PROGRAM CycleTest
VAR
	bCycleStart1:BOOL:= FALSE;
	bCycleStart2:BOOL:= FALSE;
	LevelToStart:INT:=3;
	iLevel:INT:=1;
	iNoOfLevel:INT:=4; //NO_OF_LEVEL;
	nState:INT;
	nCount:INT:=1;
	fbGUI_TEST : ARRAY [1..NO_OF_LEVEL] OF FB_GUI_TEST;
	arrLevelStartBits :ARRAY[1..NO_OF_LEVEL] OF BOOL;
	
	TDelay : TON;
	TDelay1: TON;
	TDelay2 : TON;
	ClearTCSEvent: TON;
	tCaptureDelay: TIME:= T#1000MS;
	tDelayNextStep: TIME:= T#2000MS;
	tInterval: TIME:= T#200MS;
	tempstr :STRING;
	i:INT;
	iClearCount: INT;
	iTotalClear: INT:=20;
	
	nNoOfCyclePerLevel:INT:=1;
	bStartCycle	:BOOL;
	bStart		:BOOL;
	stVIO :ST_TCMultiLevel_VIO;
	isError:BOOL;
	
	arrCount:ARRAY[1..NO_OF_LEVEL] OF INT;
	NoOfCycCount:INT :=5;
END_VAR

//<region>
	CASE nState OF
		0:
			nState:=1;
			iLevel:=LevelToStart;
		1:
			IF bCycleStart1 AND bCycleStart2 THEN 
				nState:=2; 
			ELSE
				IF bCycleStart1 XOR bCycleStart2 THEN
					bCycleStart1:=FALSE;
					bCycleStart2:=FALSE;
				END_IF
				iLevel:=LevelToStart;
			END_IF
		2:
			arrLevelStartBits[iLevel]:=TRUE;
			nState:=3;
		3:	stVIO:=arrTCMultiLevel[iLevel].fbTCMultiLevelSeq.stMLVIO;
			
			IF bCycleStart1 AND bCycleStart2 AND NOT isError THEN
				arrTCSEventTriggered :=FALSE;
				fbGUI_TEST[iLevel](iLevel:=iLevel,nCount:=nCount,bStart:=arrLevelStartBits[iLevel]);
				isError:= stVIO.isTIIError OR stVIO.isSysError OR arrTCMultiLevel[iLevel].fbTCMultiLevelSeq.P_bError;
				IF NOT arrLevelStartBits[iLevel] THEN 
					arrCount[iLevel]:=arrCount[iLevel]+1;
					Logging.fbDebugLog.M_nLogger(1, sSource:='LEVEL CYCLE COUNT', F_concat3('Level',F_concat3('[',INT_TO_STRING(iLevel), ']'), F_concat3('Cycle Count =',', ',INT_TO_STRING(arrCount[iLevel]) ) ) );
					IF iLevel < iNoOfLevel THEN
						iLevel:=iLevel+1;
						nState:=4;
					ELSIF iLevel >= iNoOfLevel THEN
						IF arrCount[iLevel]>=NoOfCycCount THEN
							arrCount[iLevel]:=0;
							bCycleStart1:=bCycleStart2 := FALSE;
						END_IF
						iLevel:=LevelToStart;
						nState:=4;
					END_IF
				END_IF	
			END_IF
			IF isError THEN
				isError:= stVIO.isTIIError OR stVIO.isSysError OR arrTCMultiLevel[iLevel].fbTCMultiLevelSeq.P_bError;
			END_IF
		4:
			nState:=1;
		5:	
		
	END_CASE
	

//</region>

(*
//<CycleTest02>
	CASE nState OF
		0:
			TDelay(IN:=FALSE);
	 		TDelay1(IN:=FALSE);
			TDelay2(IN:=FALSE);
			i:=1;
			nState:=1;
		1:
			IF bCycleStart1 AND bCycleStart2 THEN 
				nState:=2; 
			ELSE
				IF bCycleStart1 XOR bCycleStart2 THEN
					bCycleStart1:=FALSE;
					bCycleStart2:=FALSE;
				END_IF
				iLevel:=1;
			END_IF
		2:
			arrLevelStartBits[iLevel]:=TRUE;
			nState:=3;
		3:
			arrTACommands.arrTACommands[1].sLogName := CONCAT('TIUSlideOut_TESTER_LA':CONCAT('0':INT_TO_STRING(iLevel)));
			arrTACommands.arrTACommands[1].eTaskName := E_TaskName.TIUSlideOut;
			arrTACommands.arrTACommands[1].eModuleID := LEVEL_MODULE_ID[iLevel];
			arrTACommands.arrTACommands[1].bParam[1] := TRUE;
			arrTCSCommandReady:= FALSE;
			iClearCount := iTotalClear;
			
			ClearTCSEvent(IN:=(iClearCount > 0): PT:=T#100MS);
			IF ClearTCSEvent.Q THEN
				ClearTCSEvent(IN:=FALSE);
				iClearCount := iClearCount - 1;
				arrTCSEventTriggered:= FALSE;
			END_IF
			nState:=4;
		4:	
			IF arrTCMultiLevel[iLevel].stGblParam.bShuttleMoveOut =FALSE THEN
				TDelay1(IN:=TRUE:PT:=tCaptureDelay);
				IF TDelay1.Q THEN
					TDelay2(IN:=TRUE:PT:=tInterval);
					IF TDelay2.Q THEN
											
						TDelay2(IN:=FALSE);
						tempstr[1] := F_concat3('X: ': REAL_TO_STRING(aiXConverted): ': ');
						tempstr[2] := F_concat3('Y: ': REAL_TO_STRING(aiYConverted): ': ');
						tempstr[3] := F_concat3('Z: ': REAL_TO_STRING(aiZConverted): ': ');
						
						tempstr[4] := F_concat3(tempstr[1]: tempstr[2]: tempstr[3]);
						Logging.fbDebugLog.M_nLogger(1: sSource:='aisensor': F_concat3(INT_TO_STRING(i): ': ': tempstr[4]));
						i := i+1;
					END_IF
				END_IF
				TDelay(IN:=TRUE:PT:=tDelayNextStep);//after move out: delay before move in
				IF TDelay.Q THEN
					TDelay(IN:=FALSE);
					nState := 2;
				END_IF
			END_IF
		5:	//Move In
			arrTACommands.arrTACommands[1].sLogName := CONCAT('TIUSlideOut_TESTER_LA':CONCAT('0':INT_TO_STRING(iLevel)));
			arrTACommands.arrTACommands[1].eTaskName := E_TaskName.TIUSlideOut;
			arrTACommands.arrTACommands[1].eModuleID := LEVEL_MODULE_ID[iLevel];
			arrTACommands.arrTACommands[1].bParam[1] := TRUE;
			arrTCSCommandReady:= FALSE;
			iClearCount := iTotalClear;
			
			ClearTCSEvent(IN:=(iClearCount > 0): PT:=T#100MS);
			IF ClearTCSEvent.Q THEN
				ClearTCSEvent(IN:=FALSE);
				iClearCount := iClearCount - 1;
				arrTCSEventTriggered:= FALSE;
			END_IF
			nState:=4;
			nState := 6;
		6:	//
			IF arrTCMultiLevel[iLevel].stGblParam.bShuttleMoveIn=FALSE THEN
		    	TDelay(IN:=TRUE:PT:=tDelayNextStep);//after move out: delay before move in
		    	IF TDelay.Q THEN
		    		TDelay(IN:=FALSE);
		    		nState := 0;
		    		nCount := nCount +1;
		    	END_IF	 
		    END_IF
		7:  
				IF nCount> nNoOfCyclePerLevel(*AND nState =3*) THEN
		arrLevelStartBits[iLevel] := FALSE;
		bStart:=FALSE;
		nCount:=1;
		//bPBStart := FALSE;
		
	END_IF
		
		8:	
			
			IF NOT arrLevelStartBits[iLevel] THEN 
				IF iLevel < NO_OF_LEVEL THEN
					iLevel:=iLevel+1;
					nState:=4;
				ELSIF iLevel >= NO_OF_LEVEL THEN
					iLevel:=1;
					nState:=4;
				END_IF
			END_IF	
		9:
			nState:=0;
		
	END_CASE
//</CycleTest02>
*)

END_PROGRAM

(* stored: Version 1.1.0.1, ProductVersion 3.1.4022.18
   POU CycleTest: Id {af314abb-0dcf-4959-b9e7-200d5ac48c4c}, SpecialFunc None *)
